{attribute addProperty BoxType "EL2252--0000"}
{attribute addProperty Id "ActivateAT %Q*USINT81"}
{attribute addProperty CRC "62507382"}
{attribute addProperty SizeInBites "8"}
{attribute addProperty SizeInBytes "1"}
TYPE DC_Sync_Activate_03B9C976 :
STRUCT
	{attribute addProperty Name "Activate"}
	Activate AT %Q* : USINT;
END_STRUCT
END_TYPE

(* stored: Version 1.2.0.0, ProductVersion 3.1.4024.9
   DUT DC_Sync_Activate_03B9C976: Id {a2351916-42c3-4d71-934f-bb9a1b0b6823} *)
